FUNCTION_BLOCK FB_Axis_HomeToExternalForceFeedback EXTENDS FB_Axis_HomeToHardStop
VAR_INPUT
END_VAR
VAR_OUTPUT
END_VAR
VAR
	nExternalForceFeedback AT %I*		: INT;
	fConversionFactor					: REAL := 0.1; //initialized for the LinMot load cell on TVA machine
END_VAR

PROPERTY ConversionFactor : REAL
GET
ConversionFactor := fConversionFactor;
END_GET
SET
fConversionFactor := ConversionFactor;
END_SET
END_PROPERTY

METHOD HardwareUpdate : BOOL
VAR_INPUT
END_VAR
nTorqueFeedback := REAL_TO_DINT(nExternalForceFeedback * fConversionFactor);
END_METHOD

END_FUNCTION_BLOCK

(* stored: Version 1.1.0.1, ProductVersion 3.1.4024.9
   POU FB_Axis_HomeToExternalForceFeedback: Id {d4ce5353-7cf6-4f8e-9a3e-beaba89fb381}, SpecialFunc None
   Folder 01_SUPER_Overrides: Id {da597d93-edf9-4eaa-9722-be72d510bd9c}
   Property ConversionFactor: Id {b84ef6d9-9036-4d32-9cb6-f5789bf47b49}
   Get Get: Id {a3c79ef8-1f9b-4245-a57b-2404336ddd45}
   Set Set: Id {31d23ce1-a266-4180-a655-a72c0a401b89}
   Method HardwareUpdate: Id {54558ea3-ac29-4be1-9561-520c95e4860a} *)
